// TIA Portal V16 export
// export: Created 2023-03-29T11:04:42.8386657Z, ExportSetting WithDefaults, DisplayName Totally Integrated Automation Portal, DisplayVersion V16 Update 6, DisplayName TIA Portal Version Control Interface, DisplayVersion V16 Update 2, DisplayName TIA Portal Openness, DisplayVersion V16 Update 6, DisplayName STEP 7 Professional, DisplayVersion V16 Update 6, DisplayName STEP 7 Safety, DisplayVersion V16, DisplayName WinCC Advanced, DisplayVersion V16 Update 6
FUNCTION "Przełącznik żródła sygnału ciśnienia i pracy zbiorników" : Void   // FC5, LAD
TITLE = Przełącznik źródła bar
{ S7_Optimized_Access := 'TRUE' }
AUTHOR : rtecmer
VERSION : 0.1
// Funkcja przełacza sygnał z przetwornika ciśnienia zasilanie B1, tłoczenieB2 i pompownia tłoczenie B2 na wyjścia sterujące i do instancji SCADA
// Przęłączanie sygnału źródła ciśnienia zależnie od wybranej strategi: 
// 0- wyłączone, 1- Dosilanie, 2- Przetłączanie, 3- Automat, 4- Ręczne
// stored: AutoNumber true, IsIECCheckEnabled false, SetENOAutomatically false, UDAEnableTagReadback false
   VAR_TEMP
      tmp_B6 : Real;   // ciśnie czujnik B6 za zasuwą tłoczenia
      tmp_B7 : Real;   // ciśnie czujnik B7 przed zasuwą tłoczenia
      tmp_B8 : Real;   // ciśnie czujnik B8 ssanie
   END_VAR
   VAR_TEMP   // added for the SCL form of the ladder/FBD networks
      _w1 : Bool;
   END_VAR
BEGIN

REGION Network 1: Filtr Kolmana
   // "switch_kolman" - jeśli 1 to wyłączony jeśli 0 - załączony
END_REGION

REGION Network 2 (SCL): przerwa przewodu sygnałowego czujników ciśnienia
   IF "KALMAN_DB".kalman_napiecie[0] >22.0 THEN
     // błąd czujnika 
     #tmp_B6 := 0.0;
   ELSE
     #tmp_B6:= "KALMAN_DB".kalman_napiecie[0]
     ;
   END_IF;

   IF "KALMAN_DB".pomiar_napiecie[1] > 22.0THEN
     // Sbłąd czujnika
     #tmp_B7 := 0.0;
   ELSE
     #tmp_B7 := "KALMAN_DB".pomiar_napiecie[1]
     ;
   END_IF;

   IF "KALMAN_DB".kalman_napiecie[2] > 22.0 THEN
     // błąd czujnika
     #tmp_B8 := 0.0;
   ELSE
     #tmp_B8:= "KALMAN_DB".kalman_napiecie[2]
     ;
   END_IF;
END_REGION

REGION Network 3: Ciśnienie na DN225 / Ciśnienie kierunek miasto
   // Pomiar z czujnika B6 poziom "Przetłaczanie" - wylot za zasuwą
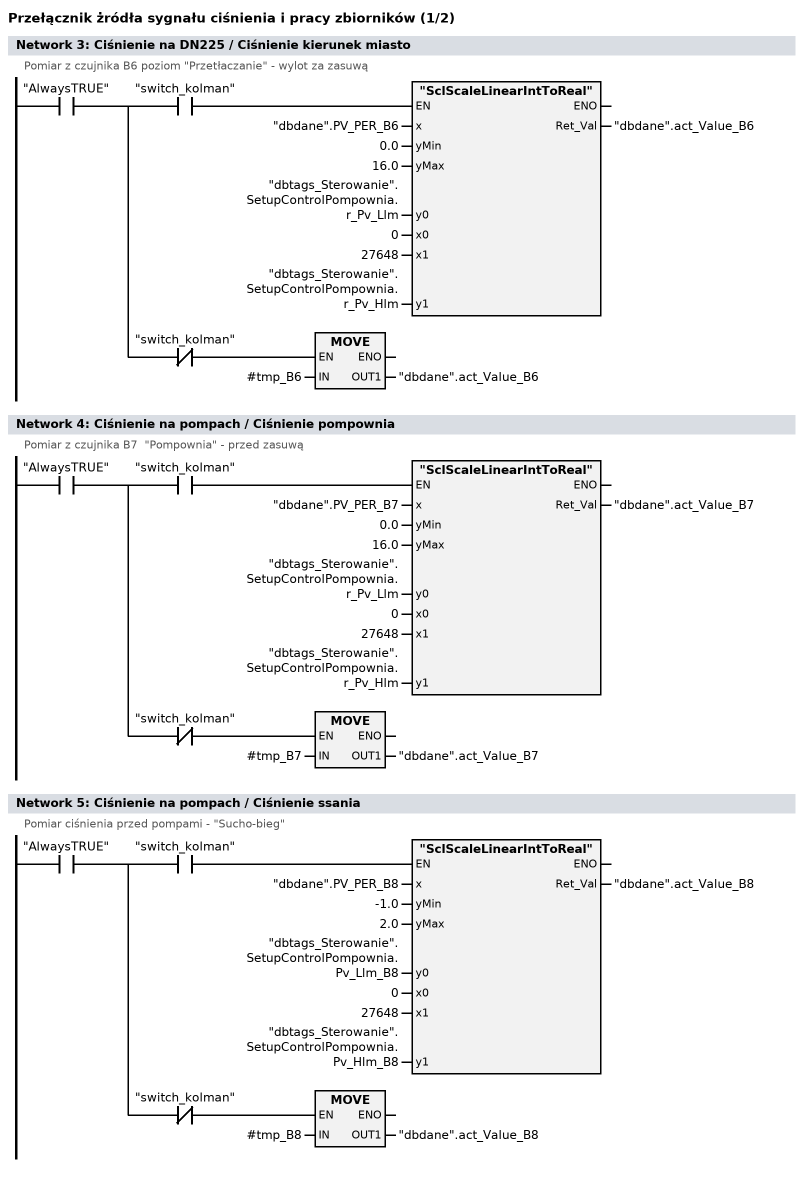
   RUNG wire#powerrail
      Contact( "AlwaysTRUE" )
      wire#w1
      Contact( "switch_kolman" )
      "SclScaleLinearIntToReal"(x := "dbdane".PV_PER_B6, yMin := 0.0, yMax := 16.0, y0 := "dbtags_Sterowanie".SetupControlPompownia.r_Pv_Llm, x0 := 0, x1 := 27648, y1 := "dbtags_Sterowanie".SetupControlPompownia.r_Pv_Hlm, Ret_Val => "dbdane".act_Value_B6)
   END_RUNG
   RUNG wire#w1
      I_Contact( "switch_kolman" )
      Move(in := #tmp_B6, out1 => "dbdane".act_Value_B6)
   END_RUNG
   // the same network as SCL:
   #_w1 := "AlwaysTRUE";
   IF "AlwaysTRUE" AND "switch_kolman" THEN
       "dbdane".act_Value_B6 := "SclScaleLinearIntToReal"(x := "dbdane".PV_PER_B6,
                               yMin := 0.0,
                               yMax := 16.0,
                               y0 := "dbtags_Sterowanie".SetupControlPompownia.r_Pv_Llm,
                               x0 := 0,
                               x1 := 27648,
                               y1 := "dbtags_Sterowanie".SetupControlPompownia.r_Pv_Hlm);
   END_IF;
   IF #_w1 AND NOT "switch_kolman" THEN "dbdane".act_Value_B6 := #tmp_B6; END_IF;
END_REGION

REGION Network 4: Ciśnienie na pompach / Ciśnienie pompownia
   // Pomiar z czujnika B7  "Pompownia" - przed zasuwą
   RUNG wire#powerrail
      Contact( "AlwaysTRUE" )
      wire#w1
      Contact( "switch_kolman" )
      "SclScaleLinearIntToReal"(x := "dbdane".PV_PER_B7, yMin := 0.0, yMax := 16.0, y0 := "dbtags_Sterowanie".SetupControlPompownia.r_Pv_Llm, x0 := 0, x1 := 27648, y1 := "dbtags_Sterowanie".SetupControlPompownia.r_Pv_Hlm, Ret_Val => "dbdane".act_Value_B7)
   END_RUNG
   RUNG wire#w1
      I_Contact( "switch_kolman" )
      Move(in := #tmp_B7, out1 => "dbdane".act_Value_B7)
   END_RUNG
   // the same network as SCL:
   #_w1 := "AlwaysTRUE";
   IF "AlwaysTRUE" AND "switch_kolman" THEN
       "dbdane".act_Value_B7 := "SclScaleLinearIntToReal"(x := "dbdane".PV_PER_B7,
                               yMin := 0.0,
                               yMax := 16.0,
                               y0 := "dbtags_Sterowanie".SetupControlPompownia.r_Pv_Llm,
                               x0 := 0,
                               x1 := 27648,
                               y1 := "dbtags_Sterowanie".SetupControlPompownia.r_Pv_Hlm);
   END_IF;
   IF #_w1 AND NOT "switch_kolman" THEN "dbdane".act_Value_B7 := #tmp_B7; END_IF;
END_REGION

REGION Network 5: Ciśnienie na pompach / Ciśnienie ssania
   // Pomiar ciśnienia przed pompami - "Sucho-bieg"
   RUNG wire#powerrail
      Contact( "AlwaysTRUE" )
      wire#w1
      Contact( "switch_kolman" )
      "SclScaleLinearIntToReal"(x := "dbdane".PV_PER_B8, yMin := -1.0, yMax := 2.0, y0 := "dbtags_Sterowanie".SetupControlPompownia.Pv_Llm_B8, x0 := 0, x1 := 27648, y1 := "dbtags_Sterowanie".SetupControlPompownia.Pv_Hlm_B8, Ret_Val => "dbdane".act_Value_B8)
   END_RUNG
   RUNG wire#w1
      I_Contact( "switch_kolman" )
      Move(in := #tmp_B8, out1 => "dbdane".act_Value_B8)
   END_RUNG
   // the same network as SCL:
   #_w1 := "AlwaysTRUE";
   IF "AlwaysTRUE" AND "switch_kolman" THEN
       "dbdane".act_Value_B8 := "SclScaleLinearIntToReal"(x := "dbdane".PV_PER_B8,
                               yMin := -1.0,
                               yMax := 2.0,
                               y0 := "dbtags_Sterowanie".SetupControlPompownia.Pv_Llm_B8,
                               x0 := 0,
                               x1 := 27648,
                               y1 := "dbtags_Sterowanie".SetupControlPompownia.Pv_Hlm_B8);
   END_IF;
   IF #_w1 AND NOT "switch_kolman" THEN "dbdane".act_Value_B8 := #tmp_B8; END_IF;
END_REGION

REGION Network 6: Wybór czujnika ciśnienia
   // Wybór czujnika pomiaru ciśnienia strategia - Dosilanie
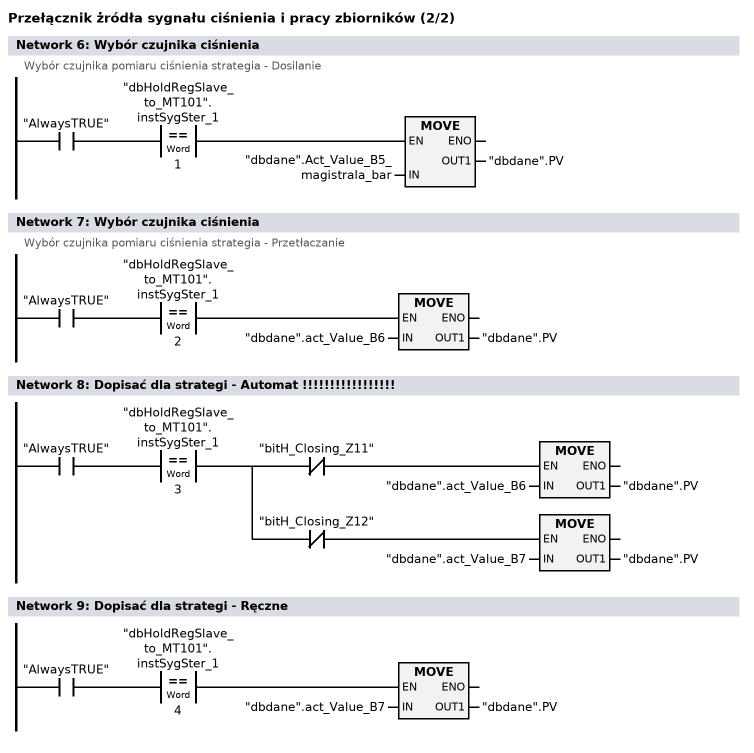
   RUNG wire#powerrail
      Contact( "AlwaysTRUE" )
      { S7_Templates := "SrcType := Word" } EQ_Contact(in1 := "dbHoldRegSlave_to_MT101".instSygSter_1, in2 := 1)
      Move(in := "dbdane".Act_Value_B5_magistrala_bar, out1 => "dbdane".PV)
   END_RUNG
   // the same network as SCL:
   IF "AlwaysTRUE" AND ("dbHoldRegSlave_to_MT101".instSygSter_1 = 1) THEN
       "dbdane".PV := "dbdane".Act_Value_B5_magistrala_bar;
   END_IF;
END_REGION

REGION Network 7: Wybór czujnika ciśnienia
   // Wybór czujnika pomiaru ciśnienia strategia - Przetłaczanie
   RUNG wire#powerrail
      Contact( "AlwaysTRUE" )
      { S7_Templates := "SrcType := Word" } EQ_Contact(in1 := "dbHoldRegSlave_to_MT101".instSygSter_1, in2 := 2)
      Move(in := "dbdane".act_Value_B6, out1 => "dbdane".PV)
   END_RUNG
   // the same network as SCL:
   IF "AlwaysTRUE" AND ("dbHoldRegSlave_to_MT101".instSygSter_1 = 2) THEN
       "dbdane".PV := "dbdane".act_Value_B6;
   END_IF;
END_REGION

REGION Network 8: Dopisać dla strategi - Automat !!!!!!!!!!!!!!!!!
   RUNG wire#powerrail
      Contact( "AlwaysTRUE" )
      { S7_Templates := "SrcType := Word" } EQ_Contact(in1 := "dbHoldRegSlave_to_MT101".instSygSter_1, in2 := 3)
      wire#w1
      I_Contact( "bitH_Closing_Z11" )
      Move(in := "dbdane".act_Value_B6, out1 => "dbdane".PV)
   END_RUNG
   RUNG wire#w1
      I_Contact( "bitH_Closing_Z12" )
      Move(in := "dbdane".act_Value_B7, out1 => "dbdane".PV)
   END_RUNG
   // the same network as SCL:
   #_w1 := "AlwaysTRUE" AND ("dbHoldRegSlave_to_MT101".instSygSter_1 = 3);
   IF #_w1 AND NOT "bitH_Closing_Z11" THEN "dbdane".PV := "dbdane".act_Value_B6; END_IF;
   IF #_w1 AND NOT "bitH_Closing_Z12" THEN "dbdane".PV := "dbdane".act_Value_B7; END_IF;
END_REGION

REGION Network 9: Dopisać dla strategi - Ręczne
   RUNG wire#powerrail
      Contact( "AlwaysTRUE" )
      { S7_Templates := "SrcType := Word" } EQ_Contact(in1 := "dbHoldRegSlave_to_MT101".instSygSter_1, in2 := 4)
      Move(in := "dbdane".act_Value_B7, out1 => "dbdane".PV)
   END_RUNG
   // the same network as SCL:
   IF "AlwaysTRUE" AND ("dbHoldRegSlave_to_MT101".instSygSter_1 = 4) THEN
       "dbdane".PV := "dbdane".act_Value_B7;
   END_IF;
END_REGION
END_FUNCTION
